(* PLC project drill, Dassault Systèmes ControlBuild 2024x *)
(* stored: creationDateTime 2023-10-03T11:13:44-01:00 *)

PROGRAM gen_panel
  VAR_OUTPUT
    powerUpPB : BOOL := false;
    startCyclePB : BOOL := false;
    emergencyStop : BOOL := false;
    batchCycle : BOOL := false;
    pieceCycle : BOOL := false;
    autoSwitch : BOOL := false;
    manualSwitch : BOOL := false;
  END_VAR
  VAR_OUTPUT
    acknowledgePB : BOOL := false;
  END_VAR

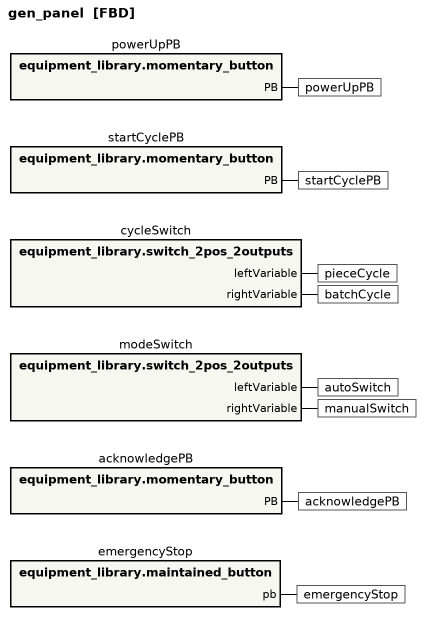
(* FBD diagram, written out as Structured Text *)
powerUpPB();
powerUpPB := powerUpPB.PB;
startCyclePB();
startCyclePB := startCyclePB.PB;
emergencyStop();
emergencyStop := emergencyStop.pb;
cycleSwitch();
pieceCycle := cycleSwitch.leftVariable;
batchCycle := cycleSwitch.rightVariable;
modeSwitch();
autoSwitch := modeSwitch.leftVariable;
manualSwitch := modeSwitch.rightVariable;
acknowledgePB();
acknowledgePB := acknowledgePB.PB;
END_PROGRAM

PROGRAM drill.drill

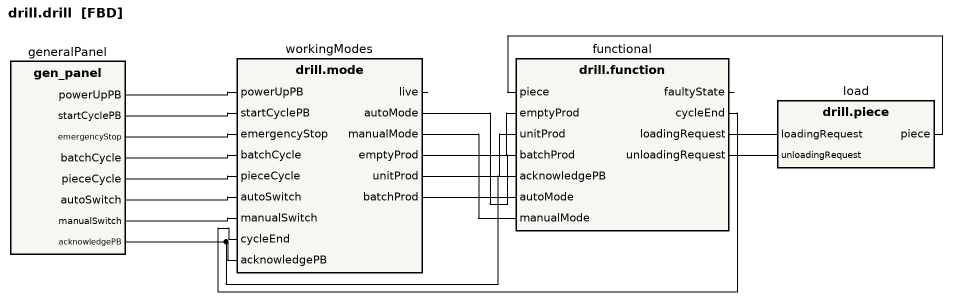
(* FBD diagram, written out as Structured Text *)
generalPanel();
load(loadingRequest := functional.loadingRequest, unloadingRequest := functional.unloadingRequest);
functional(piece := load.piece, emptyProd := workingModes.emptyProd, unitProd := workingModes.unitProd, batchProd := workingModes.batchProd, acknowledgePB := generalPanel.acknowledgePB, autoMode := workingModes.autoMode, manualMode := workingModes.manualMode);
workingModes(powerUpPB := generalPanel.powerUpPB, startCyclePB := generalPanel.startCyclePB, emergencyStop := generalPanel.emergencyStop, batchCycle := generalPanel.batchCycle, pieceCycle := generalPanel.pieceCycle, autoSwitch := generalPanel.autoSwitch, manualSwitch := generalPanel.manualSwitch, cycleEnd := functional.cycleEnd, acknowledgePB := generalPanel.acknowledgePB);
END_PROGRAM
